Universal Robots PolyScope program: empty.urp

Program empty (installation=default directory=/programs/usbdisk_1/TVT19SPL createdIn=5.11.5.1010327 lastSavedIn=5.11.5.1010327 robotSerialNumber=20195600355)
Calibrated DH parameters: a=[0.000056, -0.161146, -0.252643, 0.000052, -0.000071, 0]; d=[0.181245, -342.672485, 975.135632, -632.288651, 0.119957, 0.115765]; alpha=[1.571164, 0.001314, -0.000405, 1.570615, -1.570559, 0]; deltaTheta=[0, -1.227166, 0.434415, 0.792759, -0.000001, 0]
Robot Program (runOnlyOnce=false)
  Placeholder
